// TIA Portal project "Project2" (V17)

(* hardware
DEVICE "S7-1200 station_1"  S7-1200 Station
   slot 0: "Rack_0"  S7-1200 Rack  Rack  V1.0
   slot 1: "Master_Client"  CPU 1215C DC/DC/DC  6ES7 215-1AG40-0XB0  V4.3
DEVICE "S7-1200 station_2"  S7-1200 Station
   slot 0: "Rack_0"  S7-1200 Rack  Rack  V1.0
   slot 1: "Slave_Server"  CPU 1215C DC/DC/DC  6ES7 215-1AG40-0XB0  V4.3
DEVICE "HMI_Master"  KTP700 Basic PN
   slot 0: "HMI_Master"  KTP700 Basic PN  6AV2 123-2GB03-0AX0  15.0.0.0
   slot 1: "HMI_RT_2"  KTP700 Basic PN  6AV2 123-2GB03-0AX0  15.0.0.0
   slot 5: "HMI_Master.IE_CP_1"  PROFINET Interface  15.0.0.0
      slot 1: "PROFINET Interface_1"  PROFINET Interface
         slot 1: "Port_1"  Port
DEVICE "HMI_Slave"  KTP700 Basic PN
   slot 0: "HMI_1"  KTP700 Basic PN  6AV2 123-2GB03-0AX0  16.0.0.0
   slot 1: "HMI_RT_1"  KTP700 Basic PN  6AV2 123-2GB03-0AX0  16.0.0.0
   slot 5: "HMI_1.IE_CP_1"  PROFINET Interface  16.0.0.0
      slot 1: "PROFINET Interface_1"  PROFINET Interface
         slot 1: "Port_1"  Port
*)

// ===== PLC "Master_Client"  CPU 1215C DC/DC/DC =====

VAR_GLOBAL   // PLC tag table "Default tag table"
   "Tag_1" AT %M0.0 : Bool;
   "Tag_2" AT %Q0.3 : Bool;
   "System_Byte" AT %MB1 : Byte;
   "FirstScan" AT %M1.0 : Bool;
   "DiagStatusUpdate" AT %M1.1 : Bool;
   "AlwaysTRUE" AT %M1.2 : Bool;
   "AlwaysFALSE" AT %M1.3 : Bool;
   "Clock_Byte" AT %MB0 : Byte;
   "Clock_10Hz" AT %M0.0 : Bool;
   "Clock_5Hz" AT %M0.1 : Bool;
   "Clock_2.5Hz" AT %M0.2 : Bool;
   "Clock_2Hz" AT %M0.3 : Bool;
   "Clock_1.25Hz" AT %M0.4 : Bool;
   "Clock_1Hz" AT %M0.5 : Bool;
   "Clock_0.5Hz" AT %M0.7 : Bool;
   "Tag_6" AT %M20.0 : Bool;
   "Tag_4" AT %I0.3 : Bool;
   "Tag_5" AT %I0.4 : Bool;
   "Tag_7" AT %Q0.4 : Bool;
   "Tag_3" AT %M1.4 : Bool;
   "Tag_8" AT %M1.5 : Bool;
   "Tag_9" AT %M1.6 : Bool;
   "Tag_10" AT %M1.7 : Bool;
   "tag_1(1)" AT %MW2 : Int;
   "Tag_11" AT %M2.3 : Bool;
   "Tag_12" AT %M2.4 : Bool;
   "Tag_13" AT %M4.0 : Bool;
   "Tag_14" AT %M4.1 : Bool;
   "Tag_15" AT %M4.6 : Bool;
   "Tag_16" AT %M4.5 : Bool;
   "Tag_17" AT %M4.4 : Bool;
   "Tag_18" AT %M4.3 : Bool;
   "Tag_19" AT %M4.2 : Bool;
   "Tag_20" AT %I1.3 : Bool;
   "Tag_21" AT %M5.6 : Bool;
   "Tag_22" AT %M5.5 : Bool;
   "Tag_23" AT %M5.4 : Bool;
   "Tag_24" AT %M5.3 : Bool;
   "Tag_25" AT %M5.2 : Bool;
   "Tag_26" AT %M5.1 : Bool;
   "Tag_27" AT %M5.0 : Bool;
   "Tag_28" AT %I0.5 : Bool;
   "Tag_29" AT %Q5.5 : Bool;
   "Tag_30" AT %Q0.5 : Bool;
   "Tag_31" AT %I0.6 : Bool;
   "Tag_32" AT %Q0.6 : Bool;
   "Nhiet do vao" AT %MD5 : Real;
   "Phan hoi" AT %MD15 : Real;
   "Tag_33" AT %MD4 : DWord;
   "Tag_34" AT %I0.2 : Bool;
   "Tag_35" AT %I0.1 : Bool;
   "Tag_36" AT %I0.0 : Bool;
   "Tag_37" AT %Q0.2 : Bool;
   "Tag_38" AT %Q0.1 : Bool;
   "Tag_39" AT %Q0.0 : Bool;
   "Chuyen tiep 1" AT %QW0 : Int;
   "Chuyen tiep 2" AT %QW2 : Int;
END_VAR

DATA_BLOCK "Client_CFG_1"   // DB2
{ S7_Optimized_Access := 'FALSE' }
VERSION : 0.1
   VAR
      DISCONECT : Bool;
      MB_MODE : USInt := 1;
      MB_DATA_ADDR : UDInt := 40001;
      MB_DATA_LEN : UInt := 5;
      CONNECT : TCON_IP_v4;
      DONE : Bool;
      BUSY : Bool;
      ERROR : Bool;
      STATUS : Word;
   END_VAR
BEGIN
   CONNECT.InterfaceId := 64;
   CONNECT.ID := 1;
   CONNECT.ConnectionType := 11;
   CONNECT.ActiveEstablished := true;
   CONNECT.RemoteAddress.ADDR[1] := 192;
   CONNECT.RemoteAddress.ADDR[2] := 168;
   CONNECT.RemoteAddress.ADDR[3] := 0;
   CONNECT.RemoteAddress.ADDR[4] := 202;
   CONNECT.RemotePort := 502;
   CONNECT.LocalPort := 504;
END_DATA_BLOCK

DATA_BLOCK "Data_block_2"   // DB3
{ S7_Optimized_Access := 'FALSE' }
VERSION : 0.1
   VAR
      Data_beta : Real;
      Data1_Org : Array[0..9] of Real;
      Data2_Org : Array[0..9] of Real;
   END_VAR
BEGIN
END_DATA_BLOCK

DATA_BLOCK "Client_CFG_2"   // DB4
{ S7_Optimized_Access := 'FALSE' }
VERSION : 0.1
   VAR
      DISCONECT : Bool;
      MB_MODE : USInt := 0;
      MB_DATA_ADDR : UDInt := 40001;
      MB_DATA_LEN : UInt := 5;
      CONNECT : TCON_IP_v4;
      DONE : Bool;
      BUSY : Bool;
      ERROR : Bool;
      STATUS : Word;
   END_VAR
BEGIN
   CONNECT.InterfaceId := 64;
   CONNECT.ID := 1;
   CONNECT.ConnectionType := 11;
   CONNECT.ActiveEstablished := true;
   CONNECT.RemoteAddress.ADDR[1] := 192;
   CONNECT.RemoteAddress.ADDR[2] := 168;
   CONNECT.RemoteAddress.ADDR[3] := 0;
   CONNECT.RemoteAddress.ADDR[4] := 202;
   CONNECT.RemotePort := 502;
   CONNECT.LocalPort := 505;
END_DATA_BLOCK

FUNCTION "Word_to_bool" : Void   // FC1, LAD
{ S7_Optimized_Access := 'TRUE' }
VERSION : 0.1
   VAR_INPUT
      WORD_IN : Int;
   END_VAR
   VAR_OUTPUT
      BIT_6 : Bool;
      BIT_5 : Bool;
      BIT_4 : Bool;
      BIT_3 : Bool;
      BIT_2 : Bool;
      BIT_1 : Bool;
      BIT_0 : Bool;
   END_VAR
   VAR_TEMP
      ST_WORD : Int;
   END_VAR
BEGIN

REGION Network 1
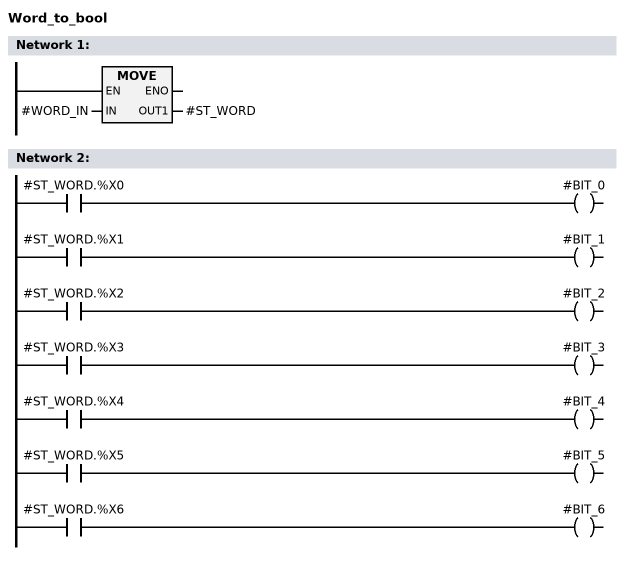
   RUNG wire#powerrail
      Move(in := #WORD_IN, out1 => #ST_WORD)
   END_RUNG
   // the same network as SCL:
   #ST_WORD := #WORD_IN;
END_REGION

REGION Network 2
   RUNG wire#powerrail
      Contact( #ST_WORD.%X0 )
      Coil( #BIT_0 )
   END_RUNG
   RUNG wire#powerrail
      Contact( #ST_WORD.%X1 )
      Coil( #BIT_1 )
   END_RUNG
   RUNG wire#powerrail
      Contact( #ST_WORD.%X2 )
      Coil( #BIT_2 )
   END_RUNG
   RUNG wire#powerrail
      Contact( #ST_WORD.%X3 )
      Coil( #BIT_3 )
   END_RUNG
   RUNG wire#powerrail
      Contact( #ST_WORD.%X4 )
      Coil( #BIT_4 )
   END_RUNG
   RUNG wire#powerrail
      Contact( #ST_WORD.%X5 )
      Coil( #BIT_5 )
   END_RUNG
   RUNG wire#powerrail
      Contact( #ST_WORD.%X6 )
      Coil( #BIT_6 )
   END_RUNG
   // the same network as SCL:
   #BIT_0 := #ST_WORD.%X0;
   #BIT_1 := #ST_WORD.%X1;
   #BIT_2 := #ST_WORD.%X2;
   #BIT_3 := #ST_WORD.%X3;
   #BIT_4 := #ST_WORD.%X4;
   #BIT_5 := #ST_WORD.%X5;
   #BIT_6 := #ST_WORD.%X6;
END_REGION
END_FUNCTION

FUNCTION "Bool_to_word" : Void   // FC2, LAD
{ S7_Optimized_Access := 'TRUE' }
VERSION : 0.1
   VAR_INPUT
      BIT_6 : Bool;
      BIT_5 : Bool;
      BIT_4 : Bool;
      BIT_3 : Bool;
      BIT_2 : Bool;
      BIT_1 : Bool;
      BIT_0 : Bool;
   END_VAR
   VAR_OUTPUT
      WORD_OUT : Int;
   END_VAR
   VAR_TEMP
      ST_WORD : Int;
   END_VAR
BEGIN

REGION Network 1
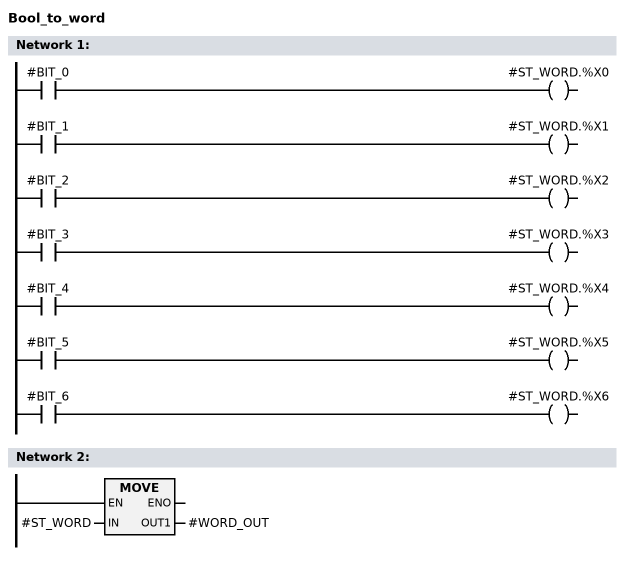
   RUNG wire#powerrail
      Contact( #BIT_0 )
      Coil( #ST_WORD.%X0 )
   END_RUNG
   RUNG wire#powerrail
      Contact( #BIT_1 )
      Coil( #ST_WORD.%X1 )
   END_RUNG
   RUNG wire#powerrail
      Contact( #BIT_2 )
      Coil( #ST_WORD.%X2 )
   END_RUNG
   RUNG wire#powerrail
      Contact( #BIT_3 )
      Coil( #ST_WORD.%X3 )
   END_RUNG
   RUNG wire#powerrail
      Contact( #BIT_4 )
      Coil( #ST_WORD.%X4 )
   END_RUNG
   RUNG wire#powerrail
      Contact( #BIT_5 )
      Coil( #ST_WORD.%X5 )
   END_RUNG
   RUNG wire#powerrail
      Contact( #BIT_6 )
      Coil( #ST_WORD.%X6 )
   END_RUNG
   // the same network as SCL:
   #ST_WORD.%X0 := #BIT_0;
   #ST_WORD.%X1 := #BIT_1;
   #ST_WORD.%X2 := #BIT_2;
   #ST_WORD.%X3 := #BIT_3;
   #ST_WORD.%X4 := #BIT_4;
   #ST_WORD.%X5 := #BIT_5;
   #ST_WORD.%X6 := #BIT_6;
END_REGION

REGION Network 2
   RUNG wire#powerrail
      Move(in := #ST_WORD, out1 => #WORD_OUT)
   END_RUNG
   // the same network as SCL:
   #WORD_OUT := #ST_WORD;
END_REGION
END_FUNCTION

ORGANIZATION_BLOCK "Write_Multi_Registers"   // OB1, LAD, ProgramCycle
TITLE = "Main Program Sweep (Cycle)"
{ S7_Optimized_Access := 'TRUE' }
VERSION : 0.1
   VAR_INPUT
      Initial_Call : Bool;   // Initial call of this OB
      Remanence : Bool;   // =True, if remanent data are available
   END_VAR
BEGIN

REGION Network 1
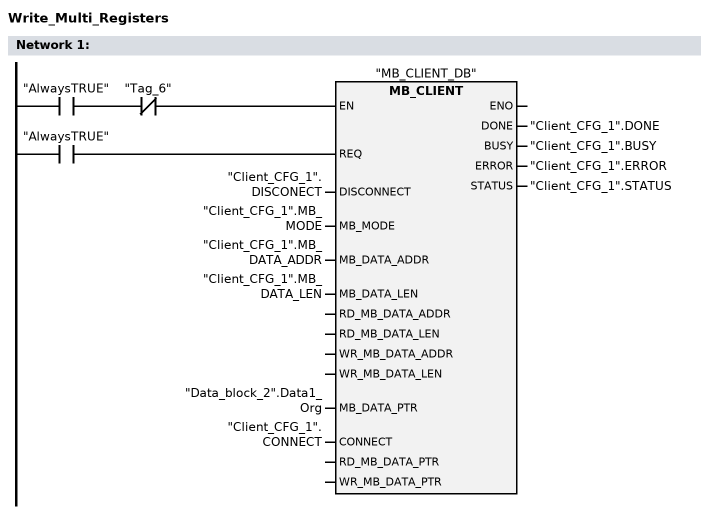
   IF "AlwaysTRUE" AND NOT "Tag_6" THEN
       "MB_CLIENT_DB"(REQ := "AlwaysTRUE",   // MB_CLIENT
                      DISCONNECT := "Client_CFG_1".DISCONECT,
                      MB_MODE := "Client_CFG_1".MB_MODE,
                      MB_DATA_ADDR := "Client_CFG_1".MB_DATA_ADDR,
                      MB_DATA_LEN := "Client_CFG_1".MB_DATA_LEN,
                      MB_DATA_PTR := "Data_block_2".Data1_Org,
                      CONNECT := "Client_CFG_1".CONNECT,
                      DONE => "Client_CFG_1".DONE,
                      BUSY => "Client_CFG_1".BUSY,
                      ERROR => "Client_CFG_1".ERROR,
                      STATUS => "Client_CFG_1".STATUS);
   END_IF;
END_REGION
END_ORGANIZATION_BLOCK

ORGANIZATION_BLOCK "Cyclic interrupt"   // OB30, LAD, CyclicInterrupt
{ S7_Optimized_Access := 'TRUE' }
VERSION : 0.1
   VAR_INPUT
      Initial_Call : Bool;   // Initial call of this OB
      Event_Count : Int;   // Events discarded
   END_VAR
BEGIN

REGION Network 1
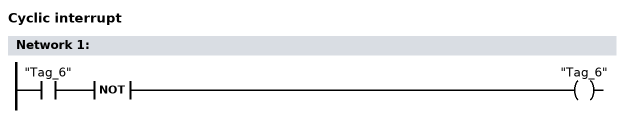
   RUNG wire#powerrail
      Contact( "Tag_6" )
      Not()
      Coil( "Tag_6" )
   END_RUNG
   // the same network as SCL:
   "Tag_6" := NOT "Tag_6";
END_REGION
END_ORGANIZATION_BLOCK

ORGANIZATION_BLOCK "Read_Multi_Registers"   // OB123, LAD, ProgramCycle
TITLE = "Main Program Sweep (Cycle)"
{ S7_Optimized_Access := 'TRUE' }
VERSION : 0.1
   VAR_INPUT
      Initial_Call : Bool;   // Initial call of this OB
      Remanence : Bool;   // =True, if remanent data are available
   END_VAR
BEGIN

REGION Network 1
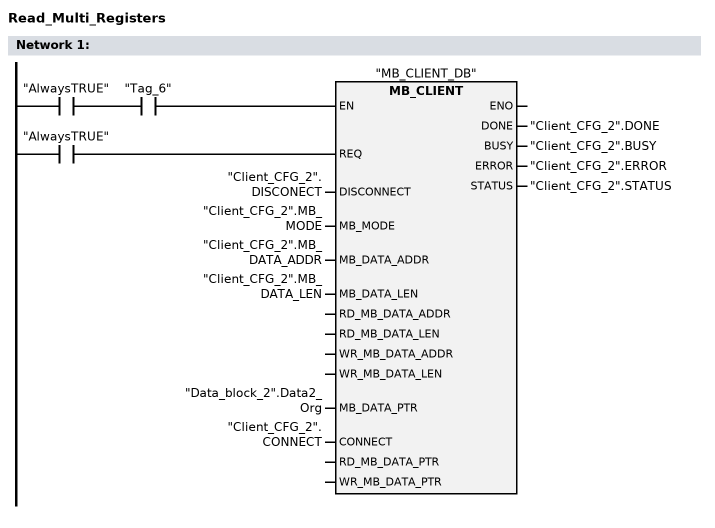
   IF "AlwaysTRUE" AND "Tag_6" THEN
       "MB_CLIENT_DB"(REQ := "AlwaysTRUE",   // MB_CLIENT
                      DISCONNECT := "Client_CFG_2".DISCONECT,
                      MB_MODE := "Client_CFG_2".MB_MODE,
                      MB_DATA_ADDR := "Client_CFG_2".MB_DATA_ADDR,
                      MB_DATA_LEN := "Client_CFG_2".MB_DATA_LEN,
                      MB_DATA_PTR := "Data_block_2".Data2_Org,
                      CONNECT := "Client_CFG_2".CONNECT,
                      DONE => "Client_CFG_2".DONE,
                      BUSY => "Client_CFG_2".BUSY,
                      ERROR => "Client_CFG_2".ERROR,
                      STATUS => "Client_CFG_2".STATUS);
   END_IF;
END_REGION
END_ORGANIZATION_BLOCK

ORGANIZATION_BLOCK "Analog"   // OB124, LAD, ProgramCycle
TITLE = "Main Program Sweep (Cycle)"
{ S7_Optimized_Access := 'TRUE' }
VERSION : 0.1
   VAR_INPUT
      Initial_Call : Bool;   // Initial call of this OB
      Remanence : Bool;   // =True, if remanent data are available
   END_VAR
BEGIN

REGION Network 1
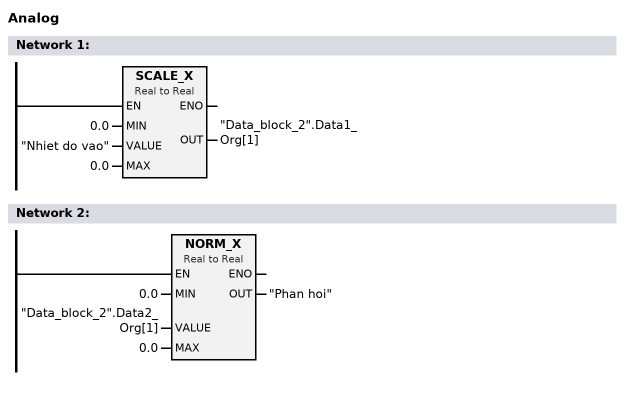
   RUNG wire#powerrail
      { S7_Templates := "[SrcType := Real, DestType := Real]" } Scale(min := 0.0, value := "Nhiet do vao", max := 0.0, out => "Data_block_2".Data1_Org[1])
   END_RUNG
   // the same network as SCL:
   "Data_block_2".Data1_Org[1] := SCALE_X(MIN := 0.0, VALUE := "Nhiet do vao", MAX := 0.0);
END_REGION

REGION Network 2
   RUNG wire#powerrail
      { S7_Templates := "[SrcType := Real, DestType := Real]" } Normalize(min := 0.0, value := "Data_block_2".Data2_Org[1], max := 0.0, out => "Phan hoi")
   END_RUNG
   // the same network as SCL:
   "Phan hoi" := NORM_X(MIN := 0.0, VALUE := "Data_block_2".Data2_Org[1], MAX := 0.0);
END_REGION
END_ORGANIZATION_BLOCK

ORGANIZATION_BLOCK "Den_master"   // OB125, LAD, ProgramCycle
TITLE = "Main Program Sweep (Cycle)"
{ S7_Optimized_Access := 'TRUE' }
VERSION : 0.1
   VAR_INPUT
      Initial_Call : Bool;   // Initial call of this OB
      Remanence : Bool;   // =True, if remanent data are available
   END_VAR
BEGIN

REGION Network 1
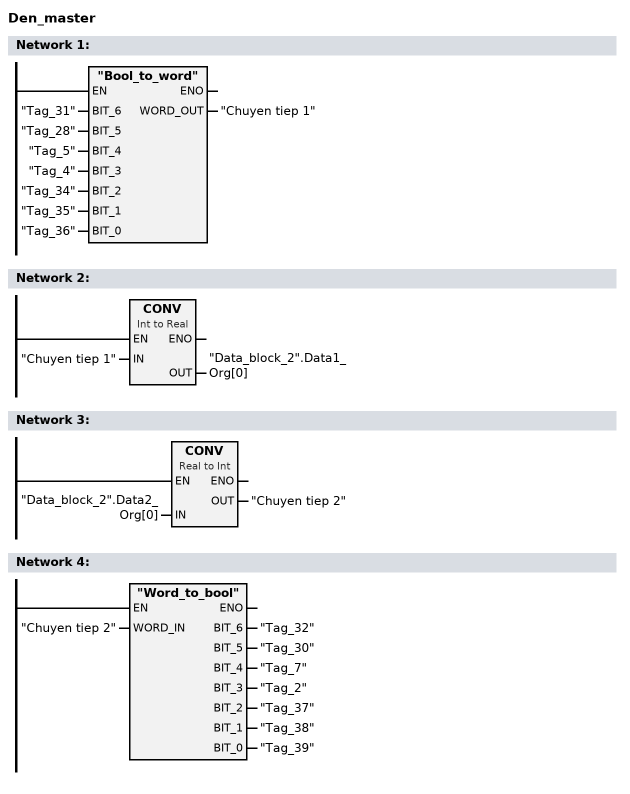
   RUNG wire#powerrail
      "Bool_to_word"(BIT_6 := "Tag_31", BIT_5 := "Tag_28", BIT_4 := "Tag_5", BIT_3 := "Tag_4", BIT_2 := "Tag_34", BIT_1 := "Tag_35", BIT_0 := "Tag_36", WORD_OUT => "Chuyen tiep 1")
   END_RUNG
   // the same network as SCL:
   "Bool_to_word"(BIT_6 := "Tag_31",
                  BIT_5 := "Tag_28",
                  BIT_4 := "Tag_5",
                  BIT_3 := "Tag_4",
                  BIT_2 := "Tag_34",
                  BIT_1 := "Tag_35",
                  BIT_0 := "Tag_36",
                  WORD_OUT => "Chuyen tiep 1");
END_REGION

REGION Network 2
   RUNG wire#powerrail
      { S7_Templates := "[SrcType := Int, DestType := Real]" } Convert(in := "Chuyen tiep 1", out => "Data_block_2".Data1_Org[0])
   END_RUNG
   // the same network as SCL:
   "Data_block_2".Data1_Org[0] := INT_TO_REAL("Chuyen tiep 1");
END_REGION

REGION Network 3
   RUNG wire#powerrail
      { S7_Templates := "[SrcType := Real, DestType := Int]" } Convert(in := "Data_block_2".Data2_Org[0], out => "Chuyen tiep 2")
   END_RUNG
   // the same network as SCL:
   "Chuyen tiep 2" := REAL_TO_INT("Data_block_2".Data2_Org[0]);
END_REGION

REGION Network 4
   RUNG wire#powerrail
      "Word_to_bool"(WORD_IN := "Chuyen tiep 2", BIT_6 => "Tag_32", BIT_5 => "Tag_30", BIT_4 => "Tag_7", BIT_3 => "Tag_2", BIT_2 => "Tag_37", BIT_1 => "Tag_38", BIT_0 => "Tag_39")
   END_RUNG
   // the same network as SCL:
   "Word_to_bool"(WORD_IN := "Chuyen tiep 2",
                  BIT_6 => "Tag_32",
                  BIT_5 => "Tag_30",
                  BIT_4 => "Tag_7",
                  BIT_3 => "Tag_2",
                  BIT_2 => "Tag_37",
                  BIT_1 => "Tag_38",
                  BIT_0 => "Tag_39");
END_REGION
END_ORGANIZATION_BLOCK

// ===== PLC "Slave_Server"  CPU 1215C DC/DC/DC =====

VAR_GLOBAL   // PLC tag table "Default tag table"
   "Tag_1" AT %I0.4 : Bool;
   "Tag_2" AT %Q0.2 : Bool;
   "System_Byte" AT %MB1 : Byte;
   "FirstScan" AT %M1.0 : Bool;
   "DiagStatusUpdate" AT %M1.1 : Bool;
   "AlwaysTRUE" AT %M1.2 : Bool;
   "AlwaysFALSE" AT %M1.3 : Bool;
   "Clock_Byte" AT %MB0 : Byte;
   "Clock_10Hz" AT %M0.0 : Bool;
   "Clock_5Hz" AT %M0.1 : Bool;
   "Clock_2.5Hz" AT %M0.2 : Bool;
   "Clock_2Hz" AT %M0.3 : Bool;
   "Clock_1.25Hz" AT %M0.4 : Bool;
   "Clock_1Hz" AT %M0.5 : Bool;
   "Clock_0.625Hz" AT %M0.6 : Bool;
   "Clock_0.5Hz" AT %M0.7 : Bool;
   "Tag_3" AT %Q0.3 : Bool;
   "Tag_4" AT %Q0.4 : Bool;
   "Tag_5" AT %M1.4 : Bool;
   "Tag_6" AT %M1.5 : Bool;
   "Tag_7" AT %M1.6 : Bool;
   "Tag_8" AT %M1.7 : Bool;
   "Tag_9" AT %M4.6 : Bool;
   "Tag_10" AT %M4.5 : Bool;
   "Tag_11" AT %M4.4 : Bool;
   "Tag_12" AT %M4.3 : Bool;
   "Tag_13" AT %M4.2 : Bool;
   "Tag_14" AT %M4.1 : Bool;
   "Tag_15" AT %M4.0 : Bool;
   "Tag_16" AT %Q4.3 : Bool;
   "Tag_17" AT %M5.3 : Bool;
   "Tag_18" AT %M5.4 : Bool;
   "Tag_19" AT %M5.6 : Bool;
   "Tag_20" AT %M5.5 : Bool;
   "Tag_21" AT %M5.2 : Bool;
   "Tag_22" AT %M5.1 : Bool;
   "Tag_23" AT %M5.0 : Bool;
   "Tag_24" AT %Q4.6 : Bool;
   "Tag_25" AT %Q0.6 : Bool;
   "Nhiet do slave" AT %MD10 : Real;
   "Tag_26" AT %MD4 : DWord;
   "chuyen tiep 1" AT %MW14 : Int;
   "chuyen tiep 2" AT %MW16 : Int;
   "Tag_27" AT %Q0.5 : Bool;
   "Tag_28" AT %Q0.1 : Bool;
   "Tag_29" AT %Q0.0 : Bool;
END_VAR

DATA_BLOCK "Server_DATA_2"   // DB1
{ S7_Optimized_Access := 'FALSE' }
VERSION : 0.1
   VAR
      DATA : Array[0..9] of Real;
      "Data Beta" : Real;
   END_VAR
BEGIN
END_DATA_BLOCK

DATA_BLOCK "Server_CFG_1"   // DB3
{ S7_Optimized_Access := 'FALSE' }
VERSION : 0.1
   VAR
      DISCONECT : Bool;
      CONNECT : TCON_IP_v4;
      NDR : Bool;
      DR : Bool;
      ERROR : Bool;
      STATUS : Word;
   END_VAR
BEGIN
   CONNECT.LocalPort := 502;
   CONNECT.RemotePort := 504;
   CONNECT.RemoteAddress.ADDR[4] := 102;
   CONNECT.RemoteAddress.ADDR[3] := 0;
   CONNECT.RemoteAddress.ADDR[2] := 168;
   CONNECT.RemoteAddress.ADDR[1] := 192;
   CONNECT.ActiveEstablished := false;
   CONNECT.ConnectionType := 11;
   CONNECT.ID := 1;
   CONNECT.InterfaceId := 64;
END_DATA_BLOCK

FUNCTION "Word_to_bool" : Void   // FC1, LAD
{ S7_Optimized_Access := 'TRUE' }
VERSION : 0.1
   VAR_INPUT
      WORD_IN : Int;
   END_VAR
   VAR_OUTPUT
      BIT_6 : Bool;
      BIT_5 : Bool;
      BIT_4 : Bool;
      BIT_3 : Bool;
      BIT_2 : Bool;
      BIT_1 : Bool;
      BIT_0 : Bool;
   END_VAR
   VAR_TEMP
      ST_WORD : Int;
   END_VAR
BEGIN

REGION Network 1
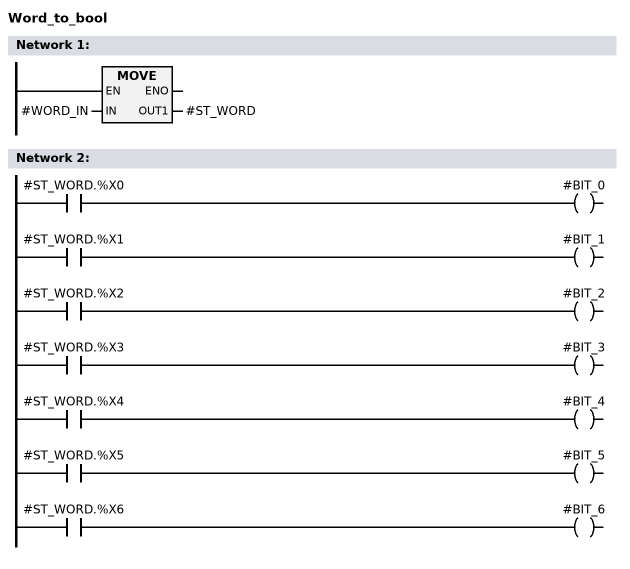
   RUNG wire#powerrail
      Move(in := #WORD_IN, out1 => #ST_WORD)
   END_RUNG
   // the same network as SCL:
   #ST_WORD := #WORD_IN;
END_REGION

REGION Network 2
   RUNG wire#powerrail
      Contact( #ST_WORD.%X0 )
      Coil( #BIT_0 )
   END_RUNG
   RUNG wire#powerrail
      Contact( #ST_WORD.%X1 )
      Coil( #BIT_1 )
   END_RUNG
   RUNG wire#powerrail
      Contact( #ST_WORD.%X2 )
      Coil( #BIT_2 )
   END_RUNG
   RUNG wire#powerrail
      Contact( #ST_WORD.%X3 )
      Coil( #BIT_3 )
   END_RUNG
   RUNG wire#powerrail
      Contact( #ST_WORD.%X4 )
      Coil( #BIT_4 )
   END_RUNG
   RUNG wire#powerrail
      Contact( #ST_WORD.%X5 )
      Coil( #BIT_5 )
   END_RUNG
   RUNG wire#powerrail
      Contact( #ST_WORD.%X6 )
      Coil( #BIT_6 )
   END_RUNG
   // the same network as SCL:
   #BIT_0 := #ST_WORD.%X0;
   #BIT_1 := #ST_WORD.%X1;
   #BIT_2 := #ST_WORD.%X2;
   #BIT_3 := #ST_WORD.%X3;
   #BIT_4 := #ST_WORD.%X4;
   #BIT_5 := #ST_WORD.%X5;
   #BIT_6 := #ST_WORD.%X6;
END_REGION
END_FUNCTION

FUNCTION "Bool_to_word" : Void   // FC2, LAD
{ S7_Optimized_Access := 'TRUE' }
VERSION : 0.1
   VAR_INPUT
      BIT_6 : Bool;
      BIT_5 : Bool;
      BIT_4 : Bool;
      BIT_3 : Bool;
      BIT_2 : Bool;
      BIT_1 : Bool;
      BIT_0 : Bool;
   END_VAR
   VAR_OUTPUT
      WORD_OUT : Int;
   END_VAR
   VAR_TEMP
      ST_WORD : Int;
   END_VAR
BEGIN

REGION Network 1
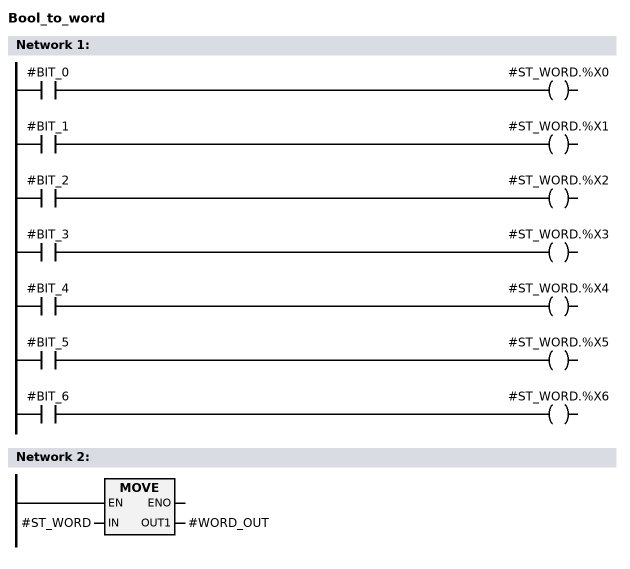
   RUNG wire#powerrail
      Contact( #BIT_0 )
      Coil( #ST_WORD.%X0 )
   END_RUNG
   RUNG wire#powerrail
      Contact( #BIT_1 )
      Coil( #ST_WORD.%X1 )
   END_RUNG
   RUNG wire#powerrail
      Contact( #BIT_2 )
      Coil( #ST_WORD.%X2 )
   END_RUNG
   RUNG wire#powerrail
      Contact( #BIT_3 )
      Coil( #ST_WORD.%X3 )
   END_RUNG
   RUNG wire#powerrail
      Contact( #BIT_4 )
      Coil( #ST_WORD.%X4 )
   END_RUNG
   RUNG wire#powerrail
      Contact( #BIT_5 )
      Coil( #ST_WORD.%X5 )
   END_RUNG
   RUNG wire#powerrail
      Contact( #BIT_6 )
      Coil( #ST_WORD.%X6 )
   END_RUNG
   // the same network as SCL:
   #ST_WORD.%X0 := #BIT_0;
   #ST_WORD.%X1 := #BIT_1;
   #ST_WORD.%X2 := #BIT_2;
   #ST_WORD.%X3 := #BIT_3;
   #ST_WORD.%X4 := #BIT_4;
   #ST_WORD.%X5 := #BIT_5;
   #ST_WORD.%X6 := #BIT_6;
END_REGION

REGION Network 2
   RUNG wire#powerrail
      Move(in := #ST_WORD, out1 => #WORD_OUT)
   END_RUNG
   // the same network as SCL:
   #WORD_OUT := #ST_WORD;
END_REGION
END_FUNCTION

ORGANIZATION_BLOCK "Main"   // OB1, LAD, ProgramCycle
TITLE = "Main Program Sweep (Cycle)"
{ S7_Optimized_Access := 'TRUE' }
VERSION : 0.1
   VAR_INPUT
      Initial_Call : Bool;   // Initial call of this OB
      Remanence : Bool;   // =True, if remanent data are available
   END_VAR
BEGIN

REGION Network 1
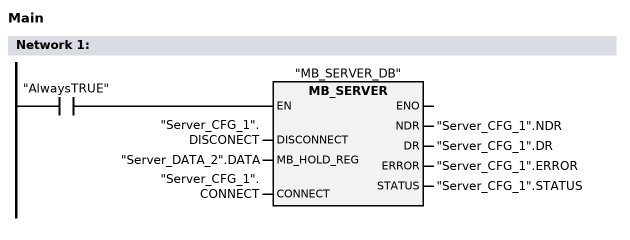
   IF "AlwaysTRUE" THEN
       "MB_SERVER_DB"(DISCONNECT := "Server_CFG_1".DISCONECT,   // MB_SERVER
                      MB_HOLD_REG := "Server_DATA_2".DATA,
                      CONNECT := "Server_CFG_1".CONNECT,
                      NDR => "Server_CFG_1".NDR,
                      DR => "Server_CFG_1".DR,
                      ERROR => "Server_CFG_1".ERROR,
                      STATUS => "Server_CFG_1".STATUS);
   END_IF;
END_REGION
END_ORGANIZATION_BLOCK

ORGANIZATION_BLOCK "Analog"   // OB123, LAD, ProgramCycle
TITLE = "Main Program Sweep (Cycle)"
{ S7_Optimized_Access := 'TRUE' }
VERSION : 0.1
   VAR_INPUT
      Initial_Call : Bool;   // Initial call of this OB
      Remanence : Bool;   // =True, if remanent data are available
   END_VAR
BEGIN

REGION Network 1
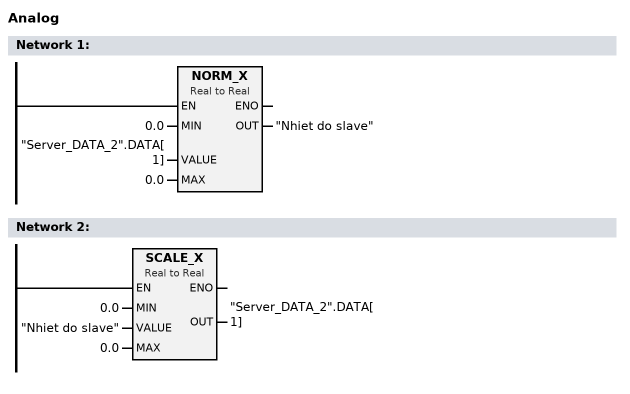
   RUNG wire#powerrail
      { S7_Templates := "[SrcType := Real, DestType := Real]" } Normalize(min := 0.0, value := "Server_DATA_2".DATA[1], max := 0.0, out => "Nhiet do slave")
   END_RUNG
   // the same network as SCL:
   "Nhiet do slave" := NORM_X(MIN := 0.0, VALUE := "Server_DATA_2".DATA[1], MAX := 0.0);
END_REGION

REGION Network 2
   RUNG wire#powerrail
      { S7_Templates := "[SrcType := Real, DestType := Real]" } Scale(min := 0.0, value := "Nhiet do slave", max := 0.0, out => "Server_DATA_2".DATA[1])
   END_RUNG
   // the same network as SCL:
   "Server_DATA_2".DATA[1] := SCALE_X(MIN := 0.0, VALUE := "Nhiet do slave", MAX := 0.0);
END_REGION
END_ORGANIZATION_BLOCK

ORGANIZATION_BLOCK "Den_slave"   // OB124, LAD, ProgramCycle
TITLE = "Main Program Sweep (Cycle)"
{ S7_Optimized_Access := 'TRUE' }
VERSION : 0.1
   VAR_INPUT
      Initial_Call : Bool;   // Initial call of this OB
      Remanence : Bool;   // =True, if remanent data are available
   END_VAR
BEGIN

REGION Network 1
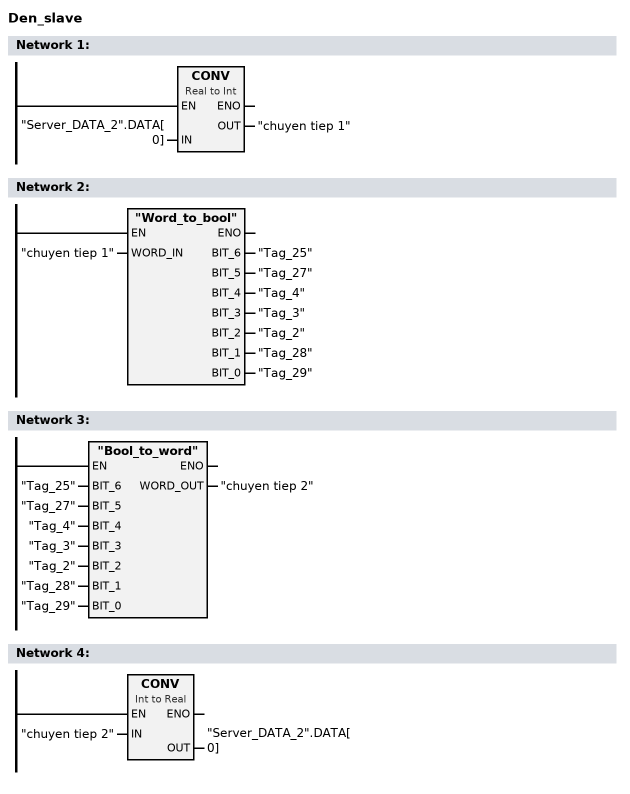
   RUNG wire#powerrail
      { S7_Templates := "[SrcType := Real, DestType := Int]" } Convert(in := "Server_DATA_2".DATA[0], out => "chuyen tiep 1")
   END_RUNG
   // the same network as SCL:
   "chuyen tiep 1" := REAL_TO_INT("Server_DATA_2".DATA[0]);
END_REGION

REGION Network 2
   RUNG wire#powerrail
      "Word_to_bool"(WORD_IN := "chuyen tiep 1", BIT_6 => "Tag_25", BIT_5 => "Tag_27", BIT_4 => "Tag_4", BIT_3 => "Tag_3", BIT_2 => "Tag_2", BIT_1 => "Tag_28", BIT_0 => "Tag_29")
   END_RUNG
   // the same network as SCL:
   "Word_to_bool"(WORD_IN := "chuyen tiep 1",
                  BIT_6 => "Tag_25",
                  BIT_5 => "Tag_27",
                  BIT_4 => "Tag_4",
                  BIT_3 => "Tag_3",
                  BIT_2 => "Tag_2",
                  BIT_1 => "Tag_28",
                  BIT_0 => "Tag_29");
END_REGION

REGION Network 3
   RUNG wire#powerrail
      "Bool_to_word"(BIT_6 := "Tag_25", BIT_5 := "Tag_27", BIT_4 := "Tag_4", BIT_3 := "Tag_3", BIT_2 := "Tag_2", BIT_1 := "Tag_28", BIT_0 := "Tag_29", WORD_OUT => "chuyen tiep 2")
   END_RUNG
   // the same network as SCL:
   "Bool_to_word"(BIT_6 := "Tag_25",
                  BIT_5 := "Tag_27",
                  BIT_4 := "Tag_4",
                  BIT_3 := "Tag_3",
                  BIT_2 := "Tag_2",
                  BIT_1 := "Tag_28",
                  BIT_0 := "Tag_29",
                  WORD_OUT => "chuyen tiep 2");
END_REGION

REGION Network 4
   RUNG wire#powerrail
      { S7_Templates := "[SrcType := Int, DestType := Real]" } Convert(in := "chuyen tiep 2", out => "Server_DATA_2".DATA[0])
   END_RUNG
   // the same network as SCL:
   "Server_DATA_2".DATA[0] := INT_TO_REAL("chuyen tiep 2");
END_REGION
END_ORGANIZATION_BLOCK

(* ===== HMI "HMI_RT_2" =====
system functions are stored by id; their names below are inferred from use
connection "HMI_Connection_3": ETHERNET, SMART_S7_1200_OMS

HMI tags "Default tag table"
   "Tag_ScreenNumber" : UInt, internal
   "Phan hoi" : Real = PLC "Phan hoi" AT %MD15, 1 s
   "Nhiet do vao" : Real = PLC "Nhiet do vao" AT %MD5, 1 s

screen "Man hinh chinh" 800x480, template "Template_1"
   on GenerateScreen: SetTag("Tag_ScreenNumber", 1)
   TextField "HmiScreenItemData" at 0,50 size 329x25; Text 'Truyền thông giá trị analog'
   Bar "Bar_1" at 547,68 size 57x334; MinimumValue 0; MaximumValue 100
      ProcessValue <- "Phan hoi"
   IOField "I/O field_1" at 107,128 size 96x32; FormatPattern s999999999.999
      ProcessValue <- "Nhiet do vao"
   TextField "HmiScreenItemData_1" at 54,160 size 207x25; Text 'Nhiệt độ gửi đi'
   TextField "HmiScreenItemData_3" at 254,158 size 207x25; Text 'Nhiệt độ phản hồi'
   IOField "I/O field_2" at 311,128 size 96x32; FormatPattern s999999999.999
      ProcessValue <- "Phan hoi"

Template "Template_1" 800x480
   Button "Exit" at 714,429 size 71x50; TextOn 'Exit'; TextOff 'Exit'; PictureOn "ExitRuntime_KTP700_Basic_PN_TR"; PictureOff "ExitRuntime_KTP700_Basic_PN_TR"
      on Release: StopRuntime(0)
   Button "Template_Button" at 614,429 size 71x50; TextOff 'Text'
   Button "Template_Button_1" at 514,429 size 71x50; TextOff 'Text'
   Button "Template_Button_2" at 414,429 size 71x50; TextOff 'Text'
   Button "Template_Button_3" at 314,429 size 71x50; TextOff 'Text'
   Button "Template_Button_4" at 214,429 size 71x50; TextOff 'Text'
   Button "Template_Button_5" at 114,429 size 71x50; TextOff 'Text'
   Button "Start screen" at 14,429 size 71x50; TextOn 'Start screen'; TextOff 'Start screen'; PictureOn "NavigateHome_KTP700_Basic_PN_TR"; PictureOff "NavigateHome_KTP700_Basic_PN_TR"
      on Release: ActivateScreen("Man hinh chinh", 0)
   SymbolicIOField "Symbolic_IO_Field_Screen" at 2,9 size 691x33; TextOn '1'; TextOff '0'; TextList "TextList_ScreenNames"
      on Change: ActivateScreenByNumber("Tag_ScreenNumber", 0)
      ProcessValue <- "Tag_ScreenNumber"
   DateTimeField "HmiScreenItemData" at 695,25 size 105x25
   DateTimeField "HmiScreenItemData_1" at 695,0 size 105x25
*)

(* ===== HMI "HMI_RT_1" =====
system functions are stored by id; their names below are inferred from use
connection "HMI_Connection_2": ETHERNET, SMART_S7_1200_OMS

HMI tags "Default tag table"
   "Tag_ScreenNumber" : UInt, internal
   "Nhiet do slave" : Real = PLC "Nhiet do slave" AT %MD10, 1 s

screen "Man hinh chinh" 800x480, template "Template_1"
   on GenerateScreen: SetTag("Tag_ScreenNumber", 1)
   TextField "HmiScreenItemData" at 0,80 size 329x25; Text 'Truyền thông giá trị analog'
   Bar "Bar_1" at 390,61 size 80x334; MinimumValue 0; MaximumValue 100
      ProcessValue <- "Nhiet do slave"
   IOField "I/O field_1" at 531,135 size 96x32; FormatPattern s999999999.999
      ProcessValue <- "Nhiet do slave"
   TextField "HmiScreenItemData_2" at 540,98 size 82x25; Text 'Nhiệt độ'

Template "Template_1" 800x480
   Button "Exit" at 714,429 size 71x50; TextOn 'Exit'; TextOff 'Exit'; PictureOn "ExitRuntime_KTP700_Basic_PN_TR"; PictureOff "ExitRuntime_KTP700_Basic_PN_TR"
      on Release: StopRuntime(0)
   Button "Template_Button" at 614,429 size 71x50; TextOff 'Text'
   Button "Template_Button_1" at 514,429 size 71x50; TextOff 'Text'
   Button "Template_Button_2" at 414,429 size 71x50; TextOff 'Text'
   Button "Template_Button_3" at 314,429 size 71x50; TextOff 'Text'
   Button "Template_Button_4" at 214,429 size 71x50; TextOff 'Text'
   Button "Template_Button_5" at 114,429 size 71x50; TextOff 'Text'
   Button "Start screen" at 14,429 size 71x50; TextOn 'Start screen'; TextOff 'Start screen'; PictureOn "NavigateHome_KTP700_Basic_PN_TR"; PictureOff "NavigateHome_KTP700_Basic_PN_TR"
      on Release: ActivateScreen("Man hinh chinh", 0)
   SymbolicIOField "Symbolic_IO_Field_Screen" at 2,9 size 691x33; TextOn '1'; TextOff '0'; TextList "TextList_ScreenNames"
      on Change: ActivateScreenByNumber("Tag_ScreenNumber", 0)
      ProcessValue <- "Tag_ScreenNumber"
   DateTimeField "HmiScreenItemData" at 695,25 size 105x25
   DateTimeField "HmiScreenItemData_1" at 695,0 size 105x25
*)